PROGRAM POU
VAR
		fbstep01:fbstepsequencer;
		step01Done:BOOL;
		step02Done:BOOL;
		step03Done:BOOL;
		step01Advance:BOOL;
		step01:stStep;
		step02:stStep;
		step03:stStep;
		iCurrentStep:INT;
END_VAR

step01.tInStepDelay:=T#10S;
step02.tInStepDelay:=T#10S;
step03.tInStepDelay:=T#10S;

fbstep01(
	iInStep:=1 , 
	iInNextStep:=2 , 
	bInStepDone:=step01.bStepDone , 
	tInStepDelay:=T#10S , 
	bInStepMode:=step01.bInStepMode , 
	bInStepAdvance:=step01.bInStepAdvance , 
	bInit:= , 
	iInitStep:= 1, 
	bOutEnterEvent=>step01.bOutEnterEvent , 
	bOutExitEvent=>step01.bOutExitEvent , 
	bOutPaused=>step01.bOutPaused, 
	iOutCurrentStep=>iCurrentStep );

	fbstep01(
	iInStep:= 2, 
	iInNextStep:=3 , 
	bInStepDone:=step02.bStepDone , 
	tInStepDelay:=T#10S , 
	bInStepMode:=step02.bInStepMode , 
	bInStepAdvance:=step02.bInStepAdvance , 
	bInit:= , 
	iInitStep:= 1, 
	bOutEnterEvent=>step02.bOutEnterEvent , 
	bOutExitEvent=>step02.bOutExitEvent , 
	bOutPaused=>step02.bOutPaused, 
	iOutCurrentStep=>iCurrentStep );

	fbstep01(
	iInStep:=3 , 
	iInNextStep:=9 , 
	bInStepDone:=step03.bStepDone , 
	tInStepDelay:=t#20s , 
	bInStepMode:=step03.bInStepMode , 
	bInStepAdvance:=step03.bInStepAdvance , 
	bInit:= , 
	iInitStep:=1 , 
	bOutEnterEvent=>step03.bOutEnterEvent , 
	bOutExitEvent=>step03.bOutExitEvent , 
	bOutPaused=>step03.bOutPaused, 
	iOutCurrentStep=>iCurrentStep );

END_PROGRAM

(* stored: Version 1.1.0.1, ProductVersion 3.1.4024.11
   POU POU: Id {66f959ed-f67b-4157-a024-45284c088de0}, SpecialFunc None *)
